(* IEC 61131-3 sources: netRob/Hardwareadapter/parser/json/functions, 3 files *)

(* ---- InitJson.ST ---- *)
(*@PROPERTIES_EX@
TYPE: POU
LOCALE: 0
IEC_LANGUAGE: ST
PLC_TYPE: independent
PROC_TYPE: independent
*)
(*@KEY@:DESCRIPTION*)

(*@KEY@:END_DESCRIPTION*)
FUNCTION InitJson : BOOL
VAR_INPUT
	input: BOOL; (* ignored *)
END_VAR
VAR_EXTERNAL
	Json: JsonConstants;
END_VAR

(*@KEY@: WORKSHEET
NAME: InitJson
IEC_LANGUAGE: ST
*)
(* JsonDataType *)
Json.Type_DOCUMENT_BEGIN := 0;
Json.Type_TYPE_STRING := 1;
Json.Type_TYPE_INTEGER := 2;
Json.Type_TYPE_DECIMAL := 3;
Json.Type_TYPE_ARRAY := 4;
Json.Type_TYPE_OBJECT := 5;
Json.Type_VALUE_TRUE := 6;
Json.Type_VALUE_FALSE := 7;
Json.Type_VALUE_NULL := 8;

(* JsonToken *)
Json.Token_BEFORE_DOCUMENT := 0;
Json.Token_AFTER_DOCUMENT := 1;
Json.Token_OPEN_OBJECT := 2; (* { *)
Json.Token_CLOSE_OBJECT := 3; (* } *)
Json.Token_OPEN_ARRAY := 4; (* [ *)
Json.Token_CLOSE_ARRAY := 5; (* ] *)
Json.Token_KEY := 6; (* " *)
Json.Token_ASSIGN := 7; (* : *)
Json.Token_VALUE := 8; (* literal *)
Json.Token_SEPARATE := 9; (* , *)

(* JsonValueParsingState *)
Json.Value_UNDEFINED := 0;
Json.Value_VALUE_STRING := 1;
Json.Value_ESCAPE := 2;
Json.Value_HEX_ESCAPE := 3;
Json.Value_BEFORE_DECIMAL := 4;
Json.Value_AFTER_DECIMAL := 5;
Json.Value_VALUE_NULL := 6;
Json.Value_VALUE_TRUE := 7;
Json.Value_VALUE_FALSE := 8;

InitJson := input;

(*@KEY@: END_WORKSHEET *)
END_FUNCTION

(* ---- JsonStream.ST ---- *)
(*@PROPERTIES_EX@
TYPE: POU
LOCALE: 0
IEC_LANGUAGE: ST
PLC_TYPE: independent
PROC_TYPE: independent
*)
(*@KEY@:DESCRIPTION*)

(*@KEY@:END_DESCRIPTION*)
FUNCTION_BLOCK JsonStream
(* Note: http://json.org/ http://notes.eatonphil.com/writing-a-simple-json-parser.html *)
VAR_IN_OUT
	(* is set by this program, when a new property is available;
		and reset by users if they wish that parsing now goes on *)
	stopForRelease: BOOL;
END_VAR
VAR_INPUT
	actualCharacter: BYTE; (* The code of the ASCII character to process next *)
END_VAR
VAR_OUTPUT
	jsonProperty: JsonProperty; (* Is only valid when stopForRelease is true *)
	parsingError: BOOL;
	parsingFinished: BOOL;
END_VAR
VAR
	parsingPosition: JsonPosition; (* logical (token based) position of the parser inside the json document *)
	newToken: BYTE (* JsonToken *);
	decreaseDepthFromLastTime: BOOL;
	increaseDepthFromLastTime: BOOL;
	insideArray: BOOL;
	insideObject: BOOL;
	nestingDepthHelper: UINT;
	debugMessage: StringKeySize;
	valueParser: JsonValueParser;
END_VAR
VAR_EXTERNAL
	Constants: GeneralConstants;
	Ascii: AsciiConstants;
	Json: JsonConstants;
END_VAR

(*@KEY@: WORKSHEET
NAME: JsonStream
IEC_LANGUAGE: ST
*)
(* Block until the caller has read the property and confirmed this by setting stopForRelease := FALSE *)
IF	stopForRelease THEN
	RETURN;
END_IF;

IF ParserGlobals.resetParser THEN (* Reset the parser *)
	parsingError := FALSE;
	parsingFinished := FALSE;
	stopForRelease := FALSE;
	parsingPosition.tokenFinished := TRUE;
	parsingPosition.actualToken := Json.Token_BEFORE_DOCUMENT;
	jsonProperty.nestingDepth := UINT#0;
	valueParser(actualCharacter := actualCharacter, newJsonToken := parsingPosition.actualToken);

	jsonProperty.nestingDepth := 0;
	jsonProperty.value.decimalValue := LREAL#0;
	jsonProperty.value.integerValue := LINT#0;
	jsonProperty.value.stringValue := '';
	jsonProperty.value.valueType := BYTE#0;
	jsonProperty.keys[1].index := UINT#0;
	jsonProperty.keys[1].propertyName := '';
	jsonProperty.keys[2].index := UINT#0;
	jsonProperty.keys[2].propertyName := '';
	jsonProperty.keys[3].index := UINT#0;
	jsonProperty.keys[3].propertyName := '';
	jsonProperty.keys[4].index := UINT#0;
	jsonProperty.keys[4].propertyName := '';
	jsonProperty.keys[5].index := UINT#0;
	jsonProperty.keys[5].propertyName := '';
	jsonProperty.keys[6].index := UINT#0;
	jsonProperty.keys[6].propertyName := '';
	jsonProperty.keys[7].index := UINT#0;
	jsonProperty.keys[7].propertyName := '';
	jsonProperty.keys[8].index := UINT#0;
	jsonProperty.keys[8].propertyName := '';
	jsonProperty.keys[9].index := UINT#0;
	jsonProperty.keys[9].propertyName := '';
	newtoken := Json.Token_BEFORE_DOCUMENT;
	insideObject := FALSE;
	nestingDepthHelper := UINT#0;
	debugMessage := 'Reset Parser';
	RETURN;
END_IF;

IF actualCharacter = Ascii.NULL
THEN
	debugMessage := 'Ascii byte is NULL';
	(* Check if buffer ended in a valid state according to json notation *)
	parsingerror := NOT(parsingPosition.actualToken = Json.Token_AFTER_DOCUMENT);
ELSE
IF NOT(parsingPosition.tokenFinished)
THEN
	debugMessage := 'Work on actual Token to finish it';
	(* WORK ON ACTUAL TOKEN TO FINISH IT *)
	valueParser(actualCharacter := actualCharacter, newJsonToken := parsingPosition.actualToken);
	(*parsingPosition.actualToken := valueParser.newJsonToken; -- Multiprog Syntax *)
	IF valueParser.resultAvailable
	THEN
		parsingPosition.tokenFinished := TRUE; (* Finish Token *)
		IF parsingPosition.actualToken = Json.Token_KEY
		THEN (* Copy token to right place *)
			nestingDepthHelper := jsonProperty.nestingDepth;
			jsonProperty.keys[nestingDepthHelper].propertyName := valueParser.result.stringValue;
		ELSE (* Release new property value *)
			(* Special cases after numbers, if end of object follows } *)
			IF parsingPosition.actualToken = Json.Token_CLOSE_OBJECT THEN
				nestingDepthHelper := jsonProperty.nestingDepth;
				IF jsonProperty.nestingDepth > UINT#0 AND
					NOT(jsonProperty.keys[nestingDepthHelper].index > UINT#00)
				THEN (* Inside object *)
					decreaseDepthFromLastTime := TRUE; (* depth will be decreased after property is read by user *)
					(* Special case: AFTER_DOCUMENT is nesting depth is 0 *)
					IF jsonProperty.nestingDepth = UINT#0 THEN
						parsingPosition.actualToken := Json.Token_AFTER_DOCUMENT;
						parsingFinished := TRUE;
					END_IF;
				ELSE
					parsingError := TRUE;
				END_IF;
			END_IF;
			(* Special cases after numbers, if end of array follows ] *)
			IF parsingPosition.actualToken = Json.Token_CLOSE_ARRAY THEN
				nestingDepthHelper := jsonProperty.nestingDepth;
				IF jsonProperty.nestingDepth = UINT#0 OR
					jsonProperty.keys[nestingDepthHelper].index = UINT#0
				THEN (* Not inside array !!! *)
					parsingError := TRUE;
				END_IF;
			END_IF;
			(* array index has already been increased at the beginning of the value *)
			jsonProperty.value := valueParser.result;
			stopForRelease := TRUE;
		END_IF;
	END_IF;
	parsingError := valueParser.parsingError; (* Error reporting *)
ELSE
IF actualCharacter <= Ascii.SPACE
THEN
	(* Whitespaces can be ignored between tokens *)
	debugMessage := 'Ignore Whitespace';
ELSE
	debugMessage := 'Validate next token: ';
	(* IF NOT A WHITESPACE AND LAST TOKEN FINISHED, VALIDATE NEXT TOKEN *)

	(* Clearup from } after number literals *)
	IF decreaseDepthFromLastTime THEN
		jsonProperty.nestingDepth := jsonProperty.nestingDepth -UINT#1;
		decreaseDepthFromLastTime := FALSE;
	END_IF;
	(* Clearup from nesting depth after { *)
	IF increaseDepthFromLastTime THEN
		jsonProperty.nestingDepth := jsonProperty.nestingDepth +UINT#1;
		increaseDepthFromLastTime := FALSE;
	END_IF;
	(* Clear up array index if array is closed *)
	IF parsingPosition.actualToken = Json.Token_CLOSE_ARRAY THEN
		nestingDepthHelper := jsonProperty.nestingDepth;
		jsonProperty.keys[nestingDepthHelper].index := UINT#0;
	END_IF;

	(* Set helper variables for actual object/appary scope *)
	insideArray := FALSE;
	insideObject := FALSE;
	IF jsonProperty.nestingDepth > UINT#0 THEN
		nestingDepthHelper := jsonProperty.nestingDepth;
		insideArray := parsingPosition.actualToken = Json.Token_OPEN_ARRAY
				OR jsonProperty.keys[nestingDepthHelper].index > UINT#0;
		insideObject := NOT(insideArray);
	END_IF;

	(* Special case: BEFORE_DOCUMENT expects } *)
	IF parsingPosition.actualToken = Json.Token_BEFORE_DOCUMENT AND actualCharacter = Ascii.OPEN_BRACE
	THEN
		debugMessage := CONCAT(debugMessage, 'OPEN_OBJECT');
		newToken := Json.Token_OPEN_OBJECT;
		(* Increase depth of nesting and clear array index flag *)
		(*lastFoundProperty.nestingDepth := lastFoundProperty.nestingDepth +UINT#1;*)
		increaseDepthFromLastTime := TRUE;
		nestingDepthHelper := jsonProperty.nestingDepth +UINT#1; (* +1 because nesting depth will be increased the next cycle *)
		jsonProperty.keys[nestingDepthHelper].index := UINT#0;
		(* Property notifiation *)
		jsonProperty.value.valueType := Json.Type_DOCUMENT_BEGIN;
		stopForRelease := TRUE;
	ELSE
	(* Valid next token is : *)
	IF actualCharacter = Ascii.COLON AND parsingPosition.actualToken = Json.Token_KEY
	THEN
		debugMessage := CONCAT(debugMessage, 'ASSIGN');
		newToken := Json.Token_ASSIGN;
	ELSE
	(* Valid next token is , *)
	IF actualCharacter = Ascii.COMMA AND (parsingPosition.actualToken = Json.Token_VALUE
			OR parsingPosition.actualToken = Json.Token_CLOSE_ARRAY
			OR (parsingPosition.actualToken = Json.Token_CLOSE_OBJECT AND (insideArray OR insideObject)))
	THEN
		debugMessage := CONCAT(debugMessage, 'SEPARATE');
		newToken := Json.Token_SEPARATE;
	ELSE
	(* Valid next token is } *)
	IF actualCharacter = Ascii.CLOSE_BRACE AND insideObject AND (parsingPosition.actualToken = Json.Token_OPEN_OBJECT
			OR parsingPosition.actualToken = Json.Token_VALUE (* Close Array and Object count as value tokens, too *)
			OR parsingPosition.actualToken = Json.Token_CLOSE_ARRAY OR parsingPosition.actualToken = Json.Token_CLOSE_OBJECT)
	THEN
		debugMessage := CONCAT(debugMessage, 'CLOSE_OBJECT');
		newToken := Json.Token_CLOSE_OBJECT;
		(* Reduce depth of nesting *)
		jsonProperty.nestingDepth := jsonProperty.nestingDepth -UINT#1;
		(* Special case: AFTER_DOCUMENT is nesting depth is 0 *)
		IF jsonProperty.nestingDepth = UINT#0 THEN
			debugMessage := CONCAT(debugMessage, 'AFTER_DOCUMENT');
			newToken := Json.Token_AFTER_DOCUMENT;
			parsingFinished := TRUE;
		END_IF;
	ELSE
	(* Valid next token is ] *)
	IF actualCharacter = Ascii.CLOSE_BRACKET AND insideArray AND (parsingPosition.actualToken = Json.Token_OPEN_ARRAY
			OR parsingPosition.actualToken = Json.Token_VALUE (* Close Array and Object count as value tokens, too *)
			OR parsingPosition.actualToken = Json.Token_CLOSE_ARRAY OR parsingPosition.actualToken = Json.Token_CLOSE_OBJECT)
	THEN
		debugMessage := CONCAT(debugMessage, 'CLOSE_ARRAY');
		newToken := Json.Token_CLOSE_ARRAY;
	ELSE
	(* Valid next token is key *)
	IF actualCharacter = Ascii.DOUBLE_QUOTE AND
			parsingPosition.actualToken = Json.Token_OPEN_OBJECT
			OR (insideObject AND parsingPosition.actualToken = Json.Token_SEPARATE)
	THEN
		debugMessage := CONCAT(debugMessage, 'KEY');
		newToken := Json.Token_KEY;
		parsingPosition.tokenFinished := FALSE;
		(* Initialising variables for string parsing (since a key is a string) *)
		valueParser(actualCharacter := actualCharacter, newJsonToken := parsingPosition.actualToken);
		(*parsingPosition.actualToken := valueParser.newJsonToken; -- Multiprog Syntax *)
		(* Result of a key token can't be finished within 1 charackter, so no check for resultAvailable *)
	ELSE
	(* Valid next token is value *)
	IF parsingPosition.actualToken = Json.Token_ASSIGN
			OR parsingPosition.actualToken = Json.Token_OPEN_ARRAY
			OR (insideArray AND parsingPosition.actualToken = Json.Token_SEPARATE)
	THEN
		debugMessage := CONCAT(debugMessage, 'VALUE');
		newToken := Json.Token_VALUE;
		parsingPosition.tokenFinished := FALSE;
		(* Initialise variables for value parsing *)
		valueParser(actualCharacter := actualCharacter, newJsonToken := parsingPosition.actualToken);
		(*parsingPosition.actualToken := valueParser.newJsonToken; -- Multiprog Syntax *)
		(* Only value tokens that can possibly be finished after 1 character are } and ] *)
		IF valueParser.resultAvailable
		THEN
			(* Release new property value *)
			parsingPosition.tokenFinished := TRUE;
			IF valueParser.result.valueType = Json.Type_TYPE_OBJECT
			THEN (* Opening Object *)
				debugMessage := CONCAT(debugMessage, 'OPEN_OBJECT');
				newToken := Json.Token_OPEN_OBJECT;
				(*lastFoundProperty.nestingDepth := lastFoundProperty.nestingDepth +UINT#1;*)
				increaseDepthFromLastTime := TRUE;
				nestingDepthHelper := jsonProperty.nestingDepth +UINT#1;(* +1 because nesting depth will be increased the next cycle *)
			ELSE (* Opening Array *)
				debugMessage := CONCAT(debugMessage, 'OPEN_ARRAY');
				newToken := Json.Token_OPEN_ARRAY;
				nestingDepthHelper := jsonProperty.nestingDepth;
			END_IF;
			jsonProperty.keys[nestingDepthHelper].index := UINT#0;
			jsonProperty.value.valueType := valueParser.result.valueType;
			stopForRelease := TRUE;
		ELSE
		nestingDepthHelper := jsonProperty.nestingDepth;
		IF NOT(valueParser.parsingError) AND (parsingPosition.actualToken = Json.Token_OPEN_ARRAY
			OR jsonProperty.keys[nestingDepthHelper].index > UINT#0)
		THEN
			(* Increase index at start of value parsing if inside array *)
			(* since Constants.JsonToken_OPEN_ARAYY will be overwritten with VALUE soon *)
			nestingDepthHelper := jsonProperty.nestingDepth;
			jsonProperty.keys[nestingDepthHelper].index :=
					jsonProperty.keys[nestingDepthHelper].index +UINT#1;
		END_IF; END_IF;
		parsingError := valueParser.parsingError; (* Error reporting *)
	ELSE
		parsingError := TRUE; (* Noting matches --> mailformed json *)
	END_IF; END_IF; END_IF; END_IF; END_IF; END_IF; END_IF;
	parsingPosition.actualToken := newToken;
END_IF; END_IF; END_IF;

(*@KEY@: END_WORKSHEET *)
END_FUNCTION_BLOCK

(* ---- JsonValueParser.ST ---- *)
(*@PROPERTIES_EX@
TYPE: POU
LOCALE: 0
IEC_LANGUAGE: ST
PLC_TYPE: independent
PROC_TYPE: independent
*)
(*@KEY@:DESCRIPTION*)

(*@KEY@:END_DESCRIPTION*)
FUNCTION_BLOCK JsonValueParser
VAR_IN_OUT
	newJsonToken: BYTE (* JsonToken *);
END_VAR
VAR_INPUT
	actualCharacter: BYTE;
END_VAR
VAR_OUTPUT
	result: JsonValue;
	resultAvailable:BOOL;
	parsingError: BOOL;
END_VAR
VAR
	valueState: BYTE (* JsonValueType *); (* := Json.Value_UNDEFINED; *)
	newValueState: BYTE (* JsonValueType *);
	alternativeCharacter: BYTE;

	stringValue: StringTextSize;
	beforeDecimal: DINT;
	afterDecimal: DINT;
	literalCounter: UINT; (* | null/true/false: position in token | number: digits after decimal point *)
	literalFlag: BOOL; (* | number: TRUE = negative number | *)
END_VAR
VAR_EXTERNAL
	Constants: GeneralConstants;
	Ascii: AsciiConstants;
	Json: JsonConstants;
END_VAR

(*@KEY@: WORKSHEET
NAME: JsonValueParser
IEC_LANGUAGE: ST
*)
(* Reset state variables *)
resultAvailable := FALSE;
parsingError := FALSE;

IF ParserGlobals.resetParser THEN
	result.decimalValue := LREAL#0;
	result.integerValue := LINT#0;
	result.stringValue := '';
	result.valueType := BYTE#0;
	stringValue := '';
	literalCounter := UINT#0;
	RETURN;
END_IF

(* Determine which value has just started *)
IF valueState = Json.Value_UNDEFINED
THEN
	IF actualCharacter = Ascii.OPEN_BRACE (* Object *) THEN
		result.valueType := Json.Type_TYPE_OBJECT;
		resultAvailable := TRUE;
	ELSE IF actualCharacter = Ascii.OPEN_BRACKET (* Array *) THEN
		result.valueType := Json.Type_TYPE_ARRAY;
		resultAvailable := TRUE;
	ELSE IF actualCharacter = Ascii.DOUBLE_QUOTE (* String *) THEN
		newValueState :=  Json.Value_VALUE_STRING;
		stringValue := '';
	ELSE IF actualCharacter = Ascii.LOWERCASE_N OR actualCharacter = Ascii.UPPERCASE_N (* null *) THEN
		newValueState :=  Json.Value_VALUE_NULL;
	ELSE IF actualCharacter = Ascii.LOWERCASE_T OR actualCharacter = Ascii.UPPERCASE_T (* true *) THEN
		newValueState :=  Json.Value_VALUE_TRUE;
	ELSE IF actualCharacter = Ascii.LOWERCASE_F OR actualCharacter = Ascii.UPPERCASE_F (* false *) THEN
		newValueState :=  Json.Value_VALUE_FALSE;
	ELSE IF actualCharacter = Ascii.PLUS OR actualCharacter = Ascii.MINUS
			OR (actualCharacter >=  Ascii.NUMBER_0 AND actualCharacter <= Ascii.NUMBER_9) (* Digit *) THEN
		newValueState :=  Json.Value_BEFORE_DECIMAL;
		beforeDecimal := DINT#0;
		afterDecimal := DINT#0;
		literalFlag := FALSE; (* positive number *)
		IF actualCharacter = Ascii.MINUS THEN
			literalFlag := TRUE; (* negative number *)
		ELSE IF NOT(actualCharacter = Ascii.PLUS) THEN (* Ignoring plus, handling numbers *)
			beforeDecimal := (BYTE_TO_DINT(actualCharacter) - BYTE_TO_DINT(Ascii.NUMBER_0));
		END_IF; END_IF;
	ELSE
			(* TODO Noting matches --> mailformed json *)
			parsingError := TRUE;
	END_IF; END_IF; END_IF; END_IF; END_IF; END_IF; END_IF;
	literalCounter := UINT#0;
ELSE
(* Work on actual (value) token to finish it *)
IF valueState = Json.Value_VALUE_STRING
THEN
	IF actualCharacter = Ascii.BACKSLASH
	THEN
		(* Skip escape character and prepare for parsing escape sequence *)
		newValueState :=  Json.Value_ESCAPE;
	ELSE
	IF actualCharacter = Ascii.DOUBLE_QUOTE
	THEN
		(* End of string value *)
		newValueState :=  Json.Value_UNDEFINED;
		result.valueType := Json.Type_TYPE_STRING;
		result.stringValue := stringValue;
		resultAvailable := TRUE;
	ELSE
	IF actualCharacter >= Ascii.SPACE
	THEN
		(* Add this character to string value and increase pointer *)
		IF LEN(stringValue) < UINT_TO_DINT(Constants.TEXT_VALUE_SIZE) THEN
			stringValue := CONCAT(stringValue, AsciiChar(actualCharacter));
		(* ELSE	*)
			(* TODO Error because things (key / string value) are too long! Or better just skip them? *)
		END_IF;
	ELSE
		(* TODO Error because non-printable character used in string *)
		parsingError := TRUE;
	END_IF; END_IF; END_IF;

ELSE
IF valueState = Json.Value_ESCAPE
THEN
	IF actualCharacter = Ascii.LOWERCASE_U
	THEN
		(* TODO prepare 4 hex digits escaping *)
		(* Actually: ignore Escape sequence and treat it as normal characters *)
		stringValue := CONCAT(stringValue, '\u');
	ELSE
		(* Single character escaping --> change actual character to whished character *)
		IF actualCharacter = Ascii.BACKSLASH OR actualCharacter = Ascii.DOUBLE_QUOTE THEN alternativeCharacter := actualCharacter; ELSE
		IF actualCharacter = Ascii.LOWERCASE_B (* backspace *) THEN alternativeCharacter := Ascii.BACKSPACE; ELSE
		IF actualCharacter = Ascii.LOWERCASE_F (* Formfeed *) THEN alternativeCharacter := Ascii.FORMFEED; ELSE
		IF actualCharacter = Ascii.LOWERCASE_N (* new line *) THEN alternativeCharacter := Ascii.NEW_LINE; ELSE
		IF actualCharacter =  Ascii.LOWERCASE_R (* carriage return *) THEN alternativeCharacter := Ascii.CARRIAGE_RETURN; ELSE
		IF actualCharacter = Ascii.LOWERCASE_T (* horizontal tab *) THEN alternativeCharacter := Ascii.HORIZONTAL_TAB; ELSE
		IF actualCharacter >= Ascii.SPACE
		THEN
			(* Add leading backslash in addition to the actual character to string value *)
			IF LEN(stringValue) < UINT_TO_DINT(Constants.TEXT_VALUE_SIZE) THEN
				stringValue := CONCAT(stringValue, '\');
			(* ELSE *)
				(* TODO Error because things (key / string value) are too long! Or better just skip them? *)
			END_IF;
		ELSE
			(* TODO Error because non-printable character used in string *)
			parsingError := TRUE;
		END_IF; END_IF; END_IF; END_IF; END_IF; END_IF; END_IF;
		(* Add (escaped) character to string value and increase pointer *)
		IF NOT(parsingError) AND LEN(stringValue) < UINT_TO_DINT(Constants.TEXT_VALUE_SIZE) THEN
			stringValue := CONCAT(stringValue, AsciiChar(alternativeCharacter));
		(* ELSE	*)
			(* TODO Error because things (key / string value) are too long! Or better just skip them? *)
		END_IF;
		newValueState := Json.Value_VALUE_STRING;
	END_IF;

ELSE
(*IF valueState = Json.Value_HEX_ESCAPE
THEN
	(* TODO *)
ELSE*)
IF valueState = Json.Value_BEFORE_DECIMAL
THEN
	IF actualCharacter = Ascii.DOT THEN
		newValueState :=  Json.Value_AFTER_DECIMAL;
		literalCounter := UINT#0;
	ELSE IF actualCharacter >= Ascii.NUMBER_0 AND actualCharacter <= Ascii.NUMBER_9 THEN
		beforeDecimal := beforeDecimal * DINT#10 + BYTE_TO_DINT(actualCharacter) - BYTE_TO_DINT(Ascii.NUMBER_0);
	ELSE IF actualCharacter = Ascii.COMMA OR actualCharacter = Ascii.CLOSE_BRACE OR actualCharacter = Ascii.CLOSE_BRACKET
			OR (actualCharacter >= Ascii.SOH AND actualCharacter <= Ascii.SPACE)
	THEN
		(* Release integer number *)
		newValueState :=  Json.Value_UNDEFINED;
		result.valueType := Json.Type_TYPE_INTEGER;
		result.integerValue := DINT_TO_INT(beforeDecimal);
		IF literalFlag THEN
			result.integerValue := -result.integerValue;
		END_IF;
		resultAvailable := TRUE;
		(* Set right next token, but JsonStream has to take care of reacting to that *)
		IF actualCharacter = Ascii.COMMA THEN
			newJsonToken := Json.Token_SEPARATE;
		ELSE IF actualCharacter = Ascii.CLOSE_BRACE THEN
			newJsonToken := Json.Token_CLOSE_OBJECT;
		ELSE IF actualCharacter = Ascii.CLOSE_BRACKET THEN
			newJsonToken := Json.Token_CLOSE_ARRAY;
		END_IF; END_IF; END_IF;
	ELSE
		(* TODO error handling *)
		parsingError := TRUE;
	END_IF; END_IF; END_IF;

ELSE
IF valueState = Json.Value_AFTER_DECIMAL
THEN
	IF actualCharacter >= Ascii.NUMBER_0 AND actualCharacter <= Ascii.NUMBER_9
	THEN
		afterDecimal := afterDecimal * 10 + actualCharacter - Ascii.NUMBER_0;
		literalCounter := literalCounter +UINT#1;
	ELSE
	IF actualCharacter = Ascii.COMMA OR actualCharacter =  Ascii.CLOSE_BRACE OR actualCharacter =  Ascii.CLOSE_BRACKET
			OR (actualCharacter >= Ascii.SOH AND actualCharacter <= Ascii.SPACE)
	THEN
		(* Release decimal number *)
		newValueState :=  Json.Value_UNDEFINED;
		result.valueType := Json.Type_TYPE_DECIMAL;
		result.decimalValue := DINT_TO_LREAL(beforeDecimal) + (DINT_TO_LREAL(afterDecimal) / EXPT(LREAL#10.0, literalCounter));
		IF literalFlag THEN
			result.decimalValue := -result.decimalValue;
		END_IF;
		resultAvailable := TRUE;
		(* Set right next token, but JsonStream has to take care of reacting to that *)
		IF actualCharacter = Ascii.COMMA THEN
			newJsonToken := Json.Token_SEPARATE;
		ELSE IF actualCharacter = Ascii.CLOSE_BRACE THEN
			newJsonToken := Json.Token_CLOSE_OBJECT;
		ELSE IF actualCharacter = Ascii.CLOSE_BRACKET THEN
			newJsonToken := Json.Token_CLOSE_ARRAY;
		END_IF; END_IF; END_IF;
	ELSE
		(* TODO error handling *)
		parsingError := TRUE;
	END_IF; END_IF;

ELSE
IF valueState = Json.Value_VALUE_NULL
THEN
	literalCounter := literalCounter + UINT#1;
	IF NOT((literalCounter = UINT#1 AND (actualCharacter = Ascii.LOWERCASE_U OR actualCharacter = Ascii.UPPERCASE_U))
			OR ((literalCounter = UINT#2 OR literalCounter = UINT#3)
			AND (actualCharacter = Ascii.LOWERCASE_L OR actualCharacter = Ascii.UPPERCASE_L)))
	THEN
		(* TODO There is an error! *)
		parsingError := TRUE;
	ELSE
	IF literalCounter = UINT#3 (* Release new property *)
	THEN
		newValueState :=  Json.Value_UNDEFINED;
		result.valueType := Json.Type_VALUE_NULL;
		resultAvailable := TRUE;
	END_IF; END_IF;

ELSE
IF valueState = Json.Value_VALUE_TRUE
THEN
	literalCounter := literalCounter +UINT#1;
	IF NOT((literalCounter = UINT#1 AND (actualCharacter = Ascii.LOWERCASE_R OR actualCharacter = Ascii.UPPERCASE_R))
			OR (literalCounter = UINT#2 AND (actualCharacter = Ascii.LOWERCASE_U OR actualCharacter = Ascii.UPPERCASE_U))
			OR (literalCounter = UINT#3 AND (actualCharacter = Ascii.LOWERCASE_E OR actualCharacter = Ascii.UPPERCASE_E)))
	THEN
		(* TODO There is an error! *)
		parsingError := TRUE;
	ELSE
	IF literalCounter = UINT#3 (* Release new property *)
	THEN
		newValueState :=  Json.Value_UNDEFINED;
		result.valueType := Json.Type_VALUE_TRUE;
		resultAvailable := TRUE;
	END_IF; END_IF;

ELSE
IF valueState = Json.Value_VALUE_FALSE
THEN
	literalCounter := literalCounter +UINT#1;
	IF NOT((literalCounter = UINT#1 AND (actualCharacter = Ascii.LOWERCASE_A OR actualCharacter = Ascii.UPPERCASE_A))
			OR (literalCounter = UINT#2 AND (actualCharacter = Ascii.LOWERCASE_L OR actualCharacter = Ascii.UPPERCASE_L))
			OR (literalCounter = UINT#3 AND (actualCharacter = Ascii.LOWERCASE_S OR actualCharacter = Ascii.UPPERCASE_S))
			OR (literalCounter = UINT#4 AND (actualCharacter = Ascii.LOWERCASE_E OR actualCharacter = Ascii.UPPERCASE_E)))
	THEN
		(* TODO There is an error! *)
		parsingError := TRUE;
	ELSE
	IF literalCounter = UINT#4 (* Release new property *)
	THEN
		newValueState :=  Json.Value_UNDEFINED;
		result.valueType := Json.Type_VALUE_FALSE;
		resultAvailable := TRUE;
	END_IF; END_IF;

END_IF; END_IF; END_IF; END_IF; END_IF; END_IF; END_IF; END_IF; (*END_IF; --> HEX_ESCAPE*)
valueState := newValueState;

(*@KEY@: END_WORKSHEET *)
END_FUNCTION_BLOCK
